PROGRAM MAIN
VAR
	//Main machine module declaration
	XPlanarModule : FB_XPlanarModule;

	//Control Source for running machine
	ControlSourceHMI : FB_ControlSource;
	ControlSourcePB	 : FB_ControlSource;

	//Local Vars
	InitComplete : BOOL;
	
	_DCLinkOK	: BOOL;
END_VAR

CyclicLogic();


// Cope Resetting Code
IF XPlanarModule.InitComplete THEN
	
	CASE XPlanarModule.CurrentState OF
		
		// Aborting - wait for rising edge of DCLinkOK
		ePMLState_aborted:
			IF XPlanarModule.DCBusOK AND NOT _DCLinkOK THEN
				XPlanarModule.ChangeState(ePMLCommand_Clear);
			END_IF

		ePMLState_Stopped:
			XPlanarModule.ChangeState(ePMLCommand_Reset);

		ePMLState_Idle:
			IF XPlanarModule._CommandedState = ePMLCommand_Clear THEN
				XPlanarModule.ChangeState(ePMLCommand_Reset);
			ELSIF XPlanarModule._CommandedState = ePMLCommand_Reset THEN
				XPlanarModule.ChangeState(ePMLCommand_Start);
			END_IF
	
	END_CASE

	// Save Previous Values
	_DCLinkOK	:= XPlanarModule.DCBusOK;
END_IF

METHOD CyclicLogic
VAR_INPUT
END_VAR
IF NOT InitComplete THEN
	InitComplete := Initialize();
	RETURN;
END_IF

//Machine support HMI & Production Monitor
ControlSourcePB.CyclicLogic();
ControlSourceHMI.CyclicLogic();

//Machine Cyclic Logic
XPlanarModule.CyclicLogic();
END_METHOD

METHOD Initialize : BOOL
//Top level machine initialization should happen here, in the main initialization METHOD. Each subsequent "layer" OF modules will be named within their respective "parent" intialize METHOD
IF NOT ControlSourceHMI.Registered THEN
	XPlanarModule.RegisterExternalController(ControlSourceHMI);
END_IF

IF NOT ControlSourcePB.Registered THEN
	XPlanarModule.RegisterExternalController(ControlSourcePB);
END_IF

ControlSourceHMI.CyclicLogic();
ControlSourcePB.CyclicLogic();

//ADSLOGSTR(ADSLOG_MSGTYPE_WARN, 'Lag Monitoring disabled', 'For simulation demo only',);
Initialize := TRUE;
END_METHOD

END_PROGRAM

(* stored: Version 1.1.0.1, ProductVersion 3.1.4026.12
   POU MAIN: Id {53f80725-e154-4e5a-96e6-b0c8fbf1d217}, SpecialFunc None
   Method CyclicLogic: Id {2e5361b9-6226-42d5-a916-4da7c200d76c}
   Method Initialize: Id {0d2644bd-d597-469b-b036-81ca046418f6} *)
